(* IEC 61131-3 sources: MotionTestBenchMaster/Logical/00_AID/AID, 2 files *)

(* ---- AID.st ---- *)
PROGRAM _CYCLIC
	FB_GetTime(enable := TRUE);
	FB_GetUtcTime(enable := TRUE);

	FB_Blink_05Hz(IN_Freq := 0.5);
	AID.DataOut.Blink05Hz	:= FB_Blink_05Hz.OUT;

	FB_Blink_1Hz(IN_Freq := 1.0);
	AID.DataOut.Blink1Hz	:= FB_Blink_1Hz.OUT;

	FB_Blink_2Hz(IN_Freq := 2.0);
	AID.DataOut.Blink2Hz	:= FB_Blink_2Hz.OUT;

	AID.DataOut.NetBlinkSlow	:= AID.DataOut.Blink1Hz;
	AID.DataOut.NetBlinkFast	:= AID.DataOut.Blink2Hz;
END_PROGRAM

(* ---- Variables.var ---- *)
VAR
	TMR_TP_HornAlarmStop : TP_Reset;
	VAR_AlarmLightReset : BOOL;
	VAR_CriticalLight : BOOL;
	VAR_AlarmLight : BOOL;
	VAR_AlarmHorn : BOOL;
	FB_Blink_05Hz : FB_Blinker;
	FB_Blink_1Hz : FB_Blinker;
	FB_Blink_2Hz : FB_Blinker;
	VAR_RedLightFix : BOOL;
	VAR_RedLightFlash : BOOL;
	VAR_BlueLightFix : BOOL;
	VAR_BlueLightFlash : BOOL;
	TMR_TON_InterCpuCycleOk : TON;
END_VAR
